SUBAPPLICATION Uebung_227_AXA (* Kombiniert 225b_AX (Dreieck-Sollwertmarker) und 226_AX (Split-Bargraph): ein Sollwert treibt beide Anzeigen, komplett über AR-Adapter-Bausteine *)
  (* Standard: 61499-2; Description: Copyright (c) 2026 Meisterschulen am Ostbahnhof This program and the accompanying materials are made available under the terms of the Eclipse Public License 2.0 which is available at https://www.eclipse.org/legal/epl-2.0/ SPDX-License-Identifier: EPL-2.0 *)
  (* Version 1.0, 2026-09-06, Franz Höpfinger, Meisterschulen am Ostbahnhof, initial API and implementation and/or initial documentation *)
  PACKAGE Uebungen;
  IMPORT Uebungen::const::UT::Dreieck::DefaultPool_Dreieck_PositionMarker::Container_PositionMarker;
  IMPORT Uebungen::const::UT::Dreieck::DefaultPool_Dreieck_BargraphSplit::Bargraph_Split_BargraphSplit;
  IMPORT Uebungen::const::UT::Dreieck::DefaultPool_Dreieck_Numeric::NumberVariable_Sollwert_N;
  IMPORT Uebungen::const::UT::Dreieck::DefaultPool_Dreieck_Numeric::NumberVariable_Istwert_N;
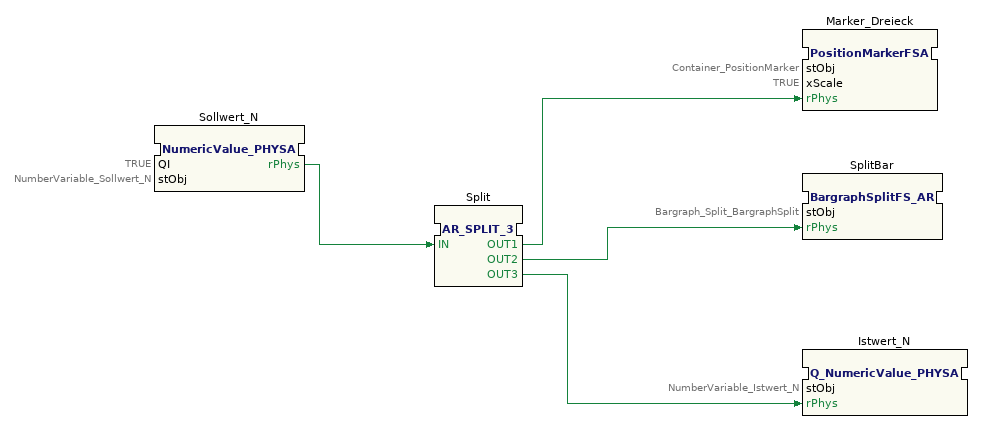
  FBS
    Sollwert_N : isobus::UT::io::NumericValue::NumericValue_PHYSA(QI := TRUE, stObj := NumberVariable_Sollwert_N);
    Split : adapter::events::unidirectional::AR_SPLIT_3;
    Marker_Dreieck : isobus::UT::Q::PositionMarkerFSA(stObj := Container_PositionMarker, xScale := TRUE);
    SplitBar : isobus::UT::Q::BargraphSplitFS_AR(stObj := Bargraph_Split_BargraphSplit);
    Istwert_N : isobus::UT::Q::Q_NumericValue_PHYSA(stObj := NumberVariable_Istwert_N);
  END_FBS
  ADAPTER_CONNECTIONS
    Sollwert_N.rPhys TO Split.IN;
    Split.OUT1 TO Marker_Dreieck.rPhys;
    Split.OUT2 TO SplitBar.rPhys;
    Split.OUT3 TO Istwert_N.rPhys;
  END_CONNECTIONS
END_SUBAPPLICATION
